// This function block is responsible for holding track of the tests and executing them.
FUNCTION_BLOCK FB_TcUnitRunner EXTENDS FB_BaseStatic
VAR
    // Indication of whether all test suites have reported that they are finished
    AllTestSuitesFinished : BOOL := FALSE;
    AllTestSuitesFinishedTrigger : R_TRIG;

    //Test result information
    TestResults : FB_TestResults;

    (* Prints the results to ADS so that Visual Studio can display the results.
       This test result formatter can be replaced with something else than ADS *)
    AdsTestResultLogger : FB_AdsTestResultLogger(TestResults);
    TestResultLogger : I_TestResultLogger := AdsTestResultLogger;

    (* If this flag is set, it means that some external event triggered the
       request to abort running the test suites *)
    AbortRunningTestSuites : BOOL;

    // Publishes a xUnit compatible XML file
    xUnitXmlPublisher : FB_xUnitXmlPublisher(TestResults);
    XmlTestResultPublisher : I_TestResultLogger := xUnitXmlPublisher;
END_VAR

(* This function sets a flag which makes the runner stop running the tests
   in the test suites *)
METHOD INTERNAL AbortRunningTestSuiteTests
AbortRunningTestSuites := TRUE;
(* Request semantics only; the runner emits 'TEST RUN ABORTED' when it honors the flag *)
TraceWithSeverity(
    Message := 'TEST RUN ABORT REQUESTED',
    Severity := Global.TcEventSeverity.Warning);
END_METHOD

// This runs all the test suites in parallel
METHOD INTERNAL RunTestSuiteTests
VAR
    Counter : UINT := 0;
    BusyPrinting : BOOL;
    (* We need to hold a temporary state of the statistics 
       as we don't consider the tests to be completely finished until all test suites have executed completely.
       The reason we want to do it this way is because a test suite can run over several cycles. Only once all tests
       are finished (which might take many cycles), do we gather correct statistics *)
    NumberOfTestSuitesFinished : UINT := 0;
END_VAR
IF GVL_TcUnit.StartedAt = 0 THEN
    GVL_TcUnit.StartedAt := F_GetCpuCounterAs64bit(GVL_TcUnit.GetCpuCounter);
    TraceWithSeverity(
        Message := CONCAT('TEST RUN STARTED - ',
                   CONCAT(UINT_TO_STRING(GVL_TcUnit.NumberOfInitializedTestSuites), ' suite(s), parallel execution')),
        Severity := Global.TcEventSeverity.Info);
END_IF

// Run TcUnit test suites
IF NOT AllTestSuitesFinished THEN
    IF GVL_TcUnit.NumberOfInitializedTestSuites = 0 THEN
        AllTestSuitesFinished := TRUE;
    ELSIF GVL_TcUnit.NumberOfInitializedTestSuites > 0 THEN
        FOR Counter := 1 TO GVL_TcUnit.NumberOfInitializedTestSuites BY 1 DO
            IF GVL_TcUnit.TestSuiteAddresses[Counter]^.AreAllTestsFinished() THEN
                NumberOfTestSuitesFinished := NumberOfTestSuitesFinished + 1;
            ELSE
                GVL_TcUnit.CurrentTestSuiteBeingCalled := GVL_TcUnit.TestSuiteAddresses[Counter];
				GVL_TcUnit.CurrentTestSuiteBeingCalled^.SetStartedAtIfNotSet(Timestamp := F_GetCpuCounterAs64bit(GVL_TcUnit.GetCpuCounter));
                GVL_TcUnit.CurrentTestSuiteBeingCalled^();
				// This is not an efficient way to set the duration
				IF GVL_TcUnit.TestSuiteAddresses[Counter]^.AreAllTestsFinished() THEN
					GVL_TcUnit.CurrentTestSuiteBeingCalled^.CalculateDuration(FinishedAt := F_GetCpuCounterAs64bit(GVL_TcUnit.GetCpuCounter));
				END_IF
            END_IF
        END_FOR
        (* Check if some event triggered an abortion of running the tests, in that case abort it now.
           This can be accomplished by setting the result of the test suites run to finished. *)
        IF AbortRunningTestSuites THEN
            (* Observed-abort effect trace: fires when the runner honors the abort flag,
               including raw online writes that never call AbortRunningTestSuiteTests().
               Naturally one-shot - the completion latch closes this branch next scan. *)
            TraceWithSeverity(
                Message := 'TEST RUN ABORTED',
                Severity := Global.TcEventSeverity.Warning);
            NumberOfTestSuitesFinished := GVL_TcUnit.NumberOfInitializedTestSuites;
        END_IF

        IF NumberOfTestSuitesFinished = GVL_TcUnit.NumberOfInitializedTestSuites THEN
            AllTestSuitesFinished := TRUE;
        END_IF
    END_IF
END_IF

AllTestSuitesFinishedTrigger(CLK := AllTestSuitesFinished);
IF AllTestSuitesFinishedTrigger.Q THEN
    TraceWithSeverity(
        Message := CONCAT('TEST RUN COMPLETED - ',
                   CONCAT(UINT_TO_STRING(GVL_TcUnit.NumberOfInitializedTestSuites), ' suite(s) finished')),
        Severity := Global.TcEventSeverity.Info);
END_IF

// Store test suite results continuously
TestResults();

// Log test suite results continuously
TestResultLogger.LogTestSuiteResults();

// Publish the xUnit Xml file once if enabled
XmlTestResultPublisher.LogTestSuiteResults();

// Run the buffered ADS logger
GVL_TcUnit.AdsMessageQueue();
END_METHOD

// This runs all the test suites in sequence (one after the other)
METHOD INTERNAL RunTestSuiteTestsInSequence
VAR_INPUT
    TimeBetweenTestSuitesExecution : TIME; // Time delay between a test suite is finished and the next test suite starts
END_VAR
VAR
    BusyPrinting : BOOL;
    (* We need to hold a temporary state of the statistics
       as we don't consider the tests to be completely finished until all test suites have executed completely.
       The reason we want to do it this way is because a test suite can run over several cycles. Only once all tests
       are finished (which might take many cycles), do we gather correct statistics *)
    NumberOfTestSuitesFinished : UINT := 0;
END_VAR
VAR_INST
    (* This variable holds which current test suite is being called, as we are running
       each one in a sequence (one by one) *)
     CurrentlyRunningTestSuite : UINT := 1;
     TimerBetweenExecutionOfTestSuites : TOF;
END_VAR
IF GVL_TcUnit.StartedAt = 0 THEN
    GVL_TcUnit.StartedAt := F_GetCpuCounterAs64bit(GVL_TcUnit.GetCpuCounter);
    TraceWithSeverity(
        Message := CONCAT('TEST RUN STARTED - ',
                   CONCAT(UINT_TO_STRING(GVL_TcUnit.NumberOfInitializedTestSuites), ' suite(s), sequential execution')),
        Severity := Global.TcEventSeverity.Info);
END_IF

TimerBetweenExecutionOfTestSuites(PT := TimeBetweenTestSuitesExecution);
// Run TcUnit test suites
IF NOT AllTestSuitesFinished THEN
    IF GVL_TcUnit.NumberOfInitializedTestSuites = 0 THEN
        AllTestSuitesFinished := TRUE;
    ELSIF GVL_TcUnit.NumberOfInitializedTestSuites > 0 THEN
        IF TimerBetweenExecutionOfTestSuites.Q THEN
            TimerBetweenExecutionOfTestSuites.IN := FALSE;
        END_IF
        IF GVL_TcUnit.TestSuiteAddresses[CurrentlyRunningTestSuite]^.AreAllTestsFinished() THEN
            IF CurrentlyRunningTestSuite <> GVL_TcUnit.NumberOfInitializedTestSuites THEN
                (* Address the finished suite directly: CurrentTestSuiteBeingCalled is
                   null until a suite has executed, e.g. when the first suite is empty *)
                GVL_TcUnit.TestSuiteAddresses[CurrentlyRunningTestSuite]^.CalculateDuration(FinishedAt := F_GetCpuCounterAs64bit(GVL_TcUnit.GetCpuCounter));
                CurrentlyRunningTestSuite := CurrentlyRunningTestSuite + 1;
                TimerBetweenExecutionOfTestSuites.IN := TRUE;
            ELSE
                (* The cursor is on the final suite and it reports finished - the whole
                   sequence is done. NumberOfTestSuitesFinished is a method VAR (reset
                   every call), so incremental counting can never reach the total; the
                   completion latch below fires from this assignment. Breadcrumb #19. *)
                NumberOfTestSuitesFinished := GVL_TcUnit.NumberOfInitializedTestSuites;
            END_IF
        ELSIF NOT TimerBetweenExecutionOfTestSuites.Q THEN
            GVL_TcUnit.CurrentTestSuiteBeingCalled := GVL_TcUnit.TestSuiteAddresses[CurrentlyRunningTestSuite];
			GVL_TcUnit.CurrentTestSuiteBeingCalled^.SetStartedAtIfNotSet(Timestamp := F_GetCpuCounterAs64bit(GVL_TcUnit.GetCpuCounter));
            GVL_TcUnit.CurrentTestSuiteBeingCalled^();
			// This is not an efficient way to set the duration
			IF GVL_TcUnit.TestSuiteAddresses[CurrentlyRunningTestSuite]^.AreAllTestsFinished() THEN
				GVL_TcUnit.CurrentTestSuiteBeingCalled^.CalculateDuration(FinishedAt := F_GetCpuCounterAs64bit(GVL_TcUnit.GetCpuCounter));
			END_IF
        END_IF
        (* Check if some event triggered an abortion of running the tests, in that case abort it now.
           This can be accomplished by setting the result of the test suites run to finished. *)
        IF AbortRunningTestSuites THEN
            (* Observed-abort effect trace: fires when the runner honors the abort flag,
               including raw online writes that never call AbortRunningTestSuiteTests().
               Naturally one-shot - the completion latch closes this branch next scan. *)
            TraceWithSeverity(
                Message := 'TEST RUN ABORTED',
                Severity := Global.TcEventSeverity.Warning);
            NumberOfTestSuitesFinished := GVL_TcUnit.NumberOfInitializedTestSuites;
        END_IF
        IF NumberOfTestSuitesFinished = GVL_TcUnit.NumberOfInitializedTestSuites THEN
            AllTestSuitesFinished := TRUE;
        END_IF
    END_IF
END_IF

AllTestSuitesFinishedTrigger(CLK := AllTestSuitesFinished);
IF AllTestSuitesFinishedTrigger.Q THEN
    TraceWithSeverity(
        Message := CONCAT('TEST RUN COMPLETED - ',
                   CONCAT(UINT_TO_STRING(GVL_TcUnit.NumberOfInitializedTestSuites), ' suite(s) finished')),
        Severity := Global.TcEventSeverity.Info);
END_IF

// Store test suite results continuously
TestResults();

// Log test suite results continuously
TestResultLogger.LogTestSuiteResults();

// Publish the xUnit Xml file once if enabled
XmlTestResultPublisher.LogTestSuiteResults();

// Run the buffered ADS logger
GVL_TcUnit.AdsMessageQueue();
END_METHOD

END_FUNCTION_BLOCK

(* stored: Version 1.1.0.1
   POU FB_TcUnitRunner: Id {857e16d6-a26c-468a-935e-aa7317c263b9}, SpecialFunc None
   Method AbortRunningTestSuiteTests: Id {3fcbd569-749a-493c-a697-2c976fa6e96a}
   Method RunTestSuiteTests: Id {d333e6c4-a1da-4b5b-91b3-4b4808e6c299}
   Method RunTestSuiteTestsInSequence: Id {01bbc2d3-b1c5-4bce-a3f3-fa46a50fd167} *)
